PROGRAM MAIN
VAR
END_VAR

END_PROGRAM

(* stored: Version 1.1.0.1
   POU MAIN: Id {d357f2d2-46b5-4ae8-b8ed-5874e6c6b56f} *)
